// Mitsubishi GX Works2 project: 2023-06-08 #3 생산자동화기능사 15번   PLC: Q03UDV
// 생산자동화기능사

// global labels: Global1
VAR_GLOBAL
  PB1 AT X0 : BOOL;
  PB2 AT X1 : BOOL;
  정지 AT X2 : BOOL;
  공급후진 AT X3 : BOOL;
  공급전진 AT X4 : BOOL;
  가공후진 AT X5 : BOOL;
  가공전진 AT X6 : BOOL;
  송출후진 AT X7 : BOOL;
  송출전진 AT X8 : BOOL;
  배출후진 AT X9 : BOOL;
  배출전진 AT X0A : BOOL;
  매거진 AT X0B : BOOL;
  금속센서 AT X0F : BOOL;
  PB3 AT X0C : BOOL;
  적 AT Y20 : BOOL;
  황 AT Y21 : BOOL;
  녹 AT Y22 : BOOL;
  공급1 AT Y23 : BOOL;
  공급2 AT Y24 : BOOL;
  가공 AT Y25 : BOOL;
  드릴 AT Y26 : BOOL;
  송출 AT Y27 : BOOL;
  배출 AT Y28 : BOOL;
  컨베이어 AT Y29 : BOOL;
END_VAR

PROGRAM 테스트동작
VAR
  PHASE : INT;
END_VAR
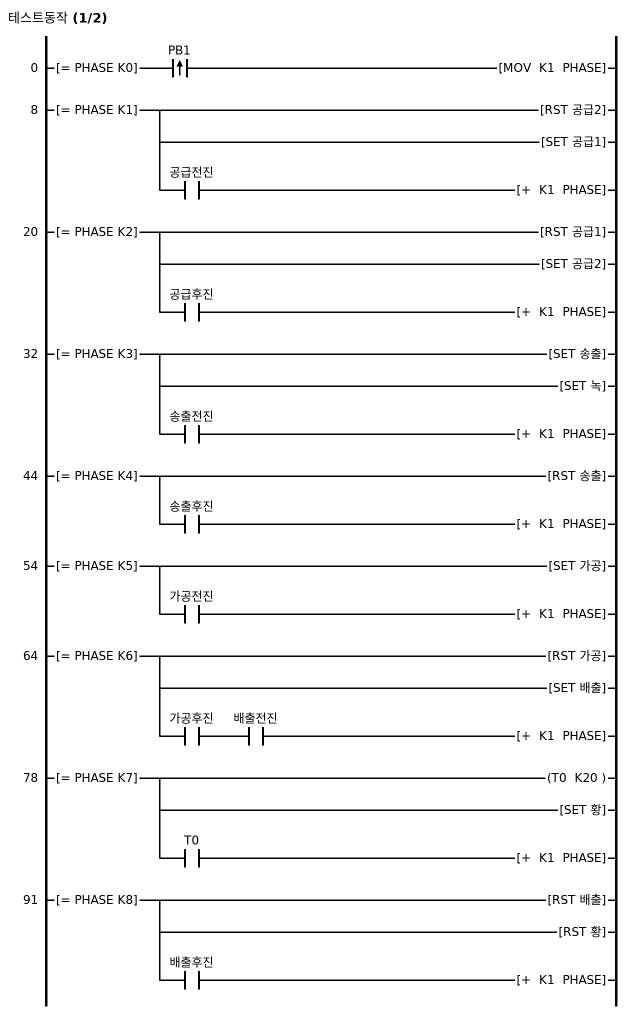
0     LD=     PHASE K0
      ANDP    PB1
      MOV     K1 PHASE
8     LD=     PHASE K1
      RST     공급2
      SET     공급1
      AND     공급전진
      +       K1 PHASE
20    LD=     PHASE K2
      RST     공급1
      SET     공급2
      AND     공급후진
      +       K1 PHASE
32    LD=     PHASE K3
      SET     송출
      SET     녹
      AND     송출전진
      +       K1 PHASE
44    LD=     PHASE K4
      RST     송출
      AND     송출후진
      +       K1 PHASE
54    LD=     PHASE K5
      SET     가공
      AND     가공전진
      +       K1 PHASE
64    LD=     PHASE K6
      RST     가공
      SET     배출
      AND     가공후진
      AND     배출전진
      +       K1 PHASE
78    LD=     PHASE K7
      OUT     T0 K20
      SET     황
      AND     T0
      +       K1 PHASE
91    LD=     PHASE K8
      RST     배출
      RST     황
      AND     배출후진
      +       K1 PHASE
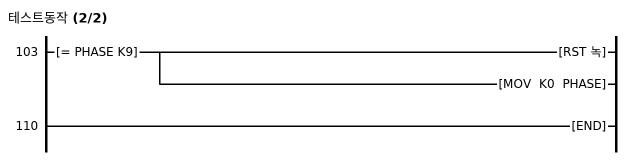
103   LD=     PHASE K9
      RST     녹
      MOV     K0 PHASE
110   END
END_PROGRAM

PROGRAM 생산자동화기능사
VAR
  PHASE : INT;
  MODE : INT;
END_VAR
VAR CONSTANT
  단속 : INT;
  연속 : INT := 1;
END_VAR
VAR
  METAL : INT;
END_VAR
VAR CONSTANT
  금속 : INT := 1;
  비금속 : INT := 2;
END_VAR
VAR
  BLINK1 : ARRAY [0..3] OF BOOL;
  BLINK2 : ARRAY [0..3] OF BOOL;
  EMIT : BOOL;
  EMG : INT;
END_VAR
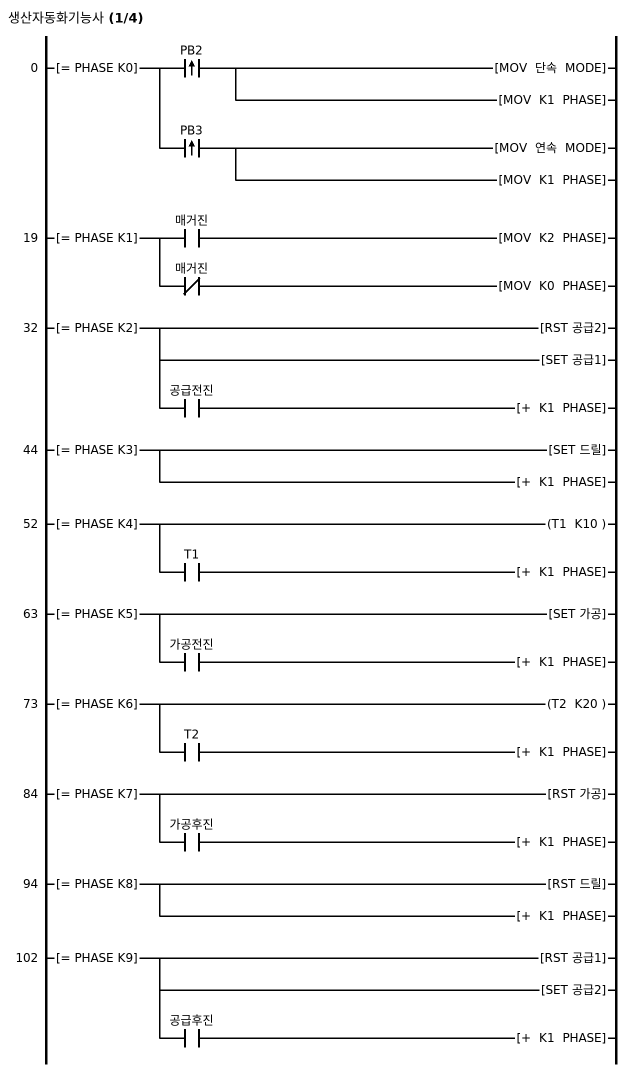
0     LD=     PHASE K0
      MPS
      ANDP    PB2
      MOV     단속 MODE
      MOV     K1 PHASE
      MPP
      ANDP    PB3
      MOV     연속 MODE
      MOV     K1 PHASE
19    LD=     PHASE K1
      MPS
      AND     매거진
      MOV     K2 PHASE
      MPP
      ANI     매거진
      MOV     K0 PHASE
32    LD=     PHASE K2
      RST     공급2
      SET     공급1
      AND     공급전진
      +       K1 PHASE
44    LD=     PHASE K3
      SET     드릴
      +       K1 PHASE
52    LD=     PHASE K4
      OUT     T1 K10
      AND     T1
      +       K1 PHASE
63    LD=     PHASE K5
      SET     가공
      AND     가공전진
      +       K1 PHASE
73    LD=     PHASE K6
      OUT     T2 K20
      AND     T2
      +       K1 PHASE
84    LD=     PHASE K7
      RST     가공
      AND     가공후진
      +       K1 PHASE
94    LD=     PHASE K8
      RST     드릴
      +       K1 PHASE
102   LD=     PHASE K9
      RST     공급1
      SET     공급2
      AND     공급후진
      +       K1 PHASE
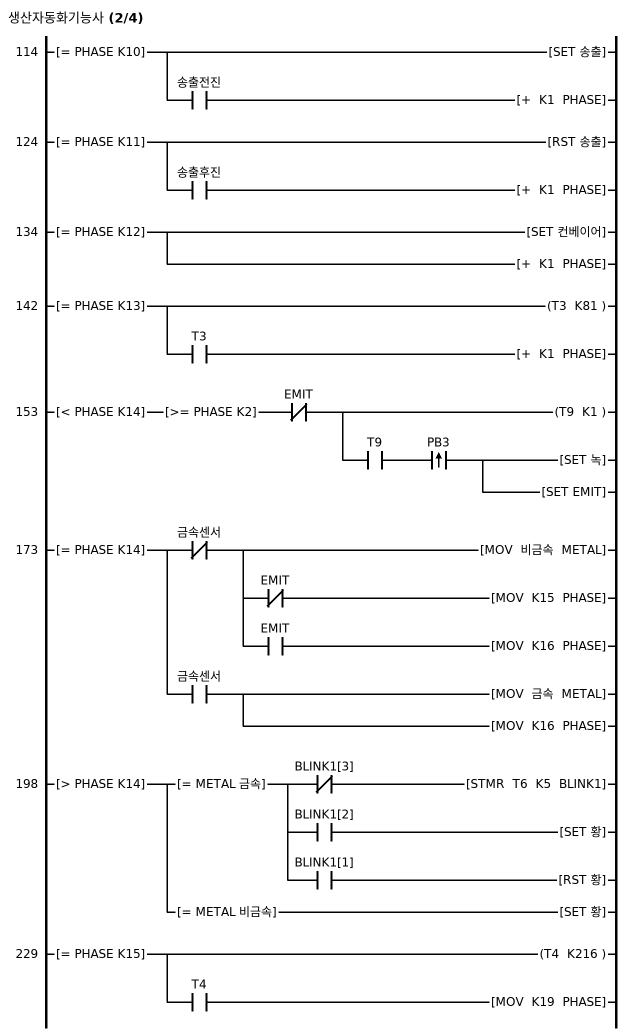
114   LD=     PHASE K10
      SET     송출
      AND     송출전진
      +       K1 PHASE
124   LD=     PHASE K11
      RST     송출
      AND     송출후진
      +       K1 PHASE
134   LD=     PHASE K12
      SET     컨베이어
      +       K1 PHASE
142   LD=     PHASE K13
      OUT     T3 K81
      AND     T3
      +       K1 PHASE
153   LD<     PHASE K14
      AND>=   PHASE K2
      ANI     EMIT
      OUT     T9 K1
      AND     T9
      ANDP    PB3
      SET     녹
      SET     EMIT
173   LD=     PHASE K14
      MPS
      ANI     금속센서
      MOV     비금속 METAL
      MPS
      ANI     EMIT
      MOV     K15 PHASE
      MPP
      AND     EMIT
      MOV     K16 PHASE
      MPP
      AND     금속센서
      MOV     금속 METAL
      MOV     K16 PHASE
198   LD>     PHASE K14
      MPS
      AND=    METAL 금속
      MPS
      ANI     BLINK1[3]
      STMR    T6 K5 BLINK1
      MRD
      AND     BLINK1[2]
      SET     황
      MPP
      AND     BLINK1[1]
      RST     황
      MPP
      AND=    METAL 비금속
      SET     황
229   LD=     PHASE K15
      OUT     T4 K216
      AND     T4
      MOV     K19 PHASE
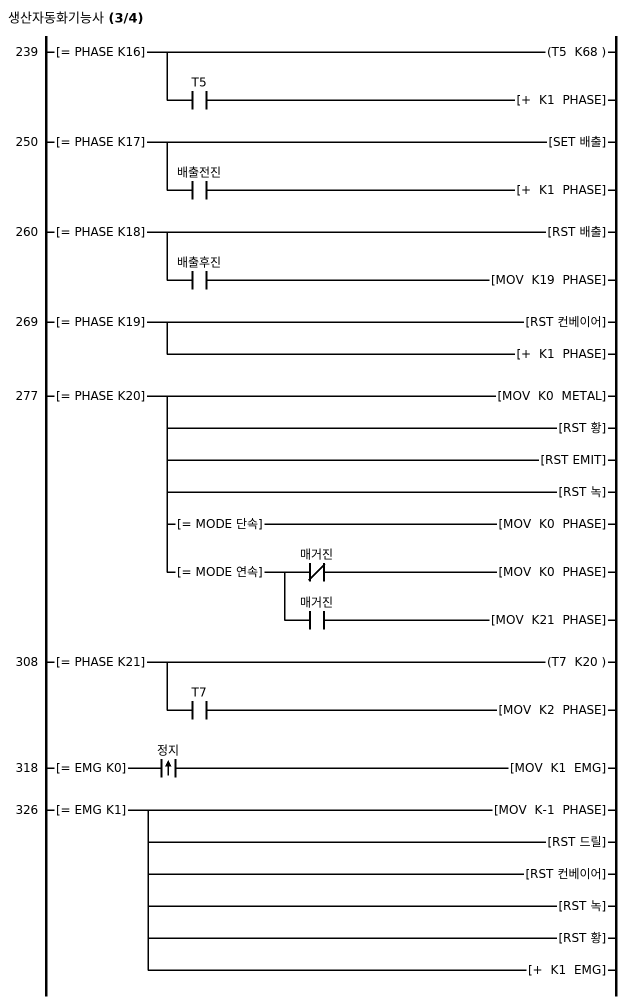
239   LD=     PHASE K16
      OUT     T5 K68
      AND     T5
      +       K1 PHASE
250   LD=     PHASE K17
      SET     배출
      AND     배출전진
      +       K1 PHASE
260   LD=     PHASE K18
      RST     배출
      AND     배출후진
      MOV     K19 PHASE
269   LD=     PHASE K19
      RST     컨베이어
      +       K1 PHASE
277   LD=     PHASE K20
      MOV     K0 METAL
      RST     황
      RST     EMIT
      RST     녹
      MPS
      AND=    MODE 단속
      MOV     K0 PHASE
      MPP
      AND=    MODE 연속
      MPS
      ANI     매거진
      MOV     K0 PHASE
      MPP
      AND     매거진
      MOV     K21 PHASE
308   LD=     PHASE K21
      OUT     T7 K20
      AND     T7
      MOV     K2 PHASE
318   LD=     EMG K0
      ANDP    정지
      MOV     K1 EMG
326   LD=     EMG K1
      MOV     K-1 PHASE
      RST     드릴
      RST     컨베이어
      RST     녹
      RST     황
      +       K1 EMG
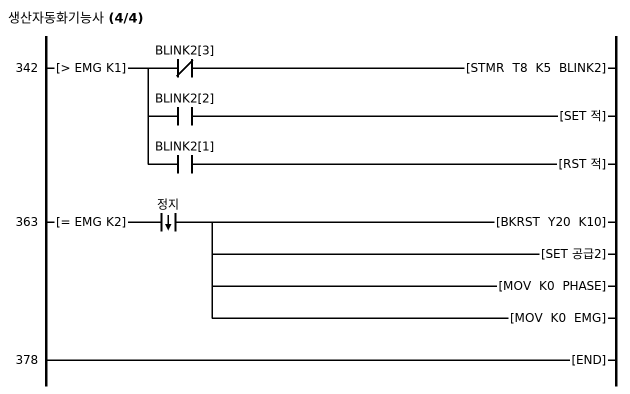
342   LD>     EMG K1
      MPS
      ANI     BLINK2[3]
      STMR    T8 K5 BLINK2
      MRD
      AND     BLINK2[2]
      SET     적
      MPP
      AND     BLINK2[1]
      RST     적
363   LD=     EMG K2
      ANDF    정지
      BKRST   Y20 K10
      SET     공급2
      MOV     K0 PHASE
      MOV     K0 EMG
378   END
END_PROGRAM
